INTERFACE I_HomingBuilder EXTENDS __System.IQueryInterface

METHOD BuildForceCalibrationCommand : I_HomingCommand
END_METHOD

METHOD BuildResetCalibrationCommand : I_HomingCommand
END_METHOD

METHOD Position : I_PositioningHomingBuilder
VAR_INPUT
	value : LREAL;
END_VAR
END_METHOD

END_INTERFACE

(* stored: Version 1.1.0.1, ProductVersion 3.1.4024.12
   Itf I_HomingBuilder: Id {c7c0e189-3799-4de7-baab-b5aa1f5a5ed5}
   Method BuildForceCalibrationCommand: Id {d843cfe5-40be-42cf-bb40-31e403e80318}
   Method BuildResetCalibrationCommand: Id {7bedc5a7-a0ff-4800-98f6-d15108cdbf2f}
   Method Position: Id {b6708fda-0bbd-4f0b-9cb1-7783ab81a7ab} *)
